(* LS Electric XG5000 project: 06_Practice7_convert_value *)
(* PLC LSPLC *)

PROGRAM NewProgram (* task: 스캔 프로그램 *)
VAR
    결과1 : INT;
    결과1_R : REAL;
    숫자1 : INT;
    숫자1_R : REAL;
END_VAR

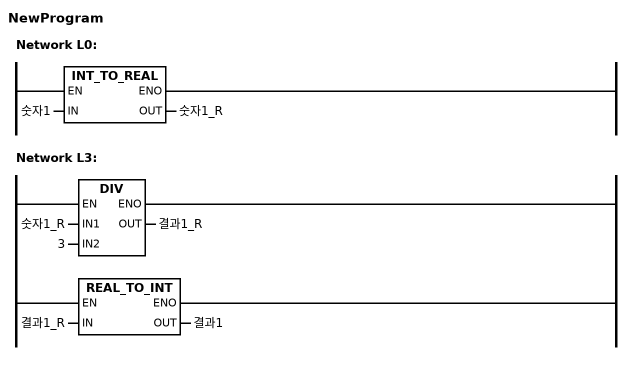
(* Rung L0 *)
숫자1_R := INT_TO_REAL(숫자1);
(* Rung L3 *)
결과1_R := 숫자1_R / 3;
결과1 := REAL_TO_INT(결과1_R);
END_PROGRAM